// Brief: Master Arm Home Posture
FUNCTION_BLOCK PUBLIC FB_StateCtrlHome EXTENDS FB_MasterArmCtrlBase
VAR_INPUT
END_VAR
VAR_OUTPUT
END_VAR
VAR
	m_homePlanner : FB_TrajMoveJ;
	
	// home motion parameters
	m_homePosture:ARRAY [1..2, 1..7] OF LREAL:=[0.0, -PI/2, 0, -PI, PI, -PI/2, 0,
							 			  			0.0, -PI/2, 0, 0, PI, PI/2, 0];
	m_homeMaxjntVel:Vec7d:=[1.0, 1.0, 1.0, 1.0, 1.0, 1.0, 1.0];
	m_homeMaxjntAcc:Vec7d:=[1.0, 1.0, 1.0, 2.0, 2.0, 2.0, 2.0];
	m_homeMaxjntJerk:Vec7d:=[7(4.0)];
	
	m_endJntPos : Vec7d;
END_VAR

// override this function in each exact controller
METHOD PROTECTED calcCmdJntPos : BOOL
VAR_IN_OUT CONSTANT
	i_slaveIdx :INT;
	i_shoulderPose :ST_Frame;
	i_masterArm :FB_MasterArm;
	i_slaveStatus :ST_SlaveStatus;
END_VAR
VAR 
	i :INT;
	curJntVel :Vec7d;
	curJntPos :Vec7d;
	posErr:Vec7d;
END_VAR
// check if planner is ready
IF m_homePlanner.isGene = FALSE THEN
	calcCmdJntPos:=FALSE;
	RETURN;
END_IF

// traj plan
calcCmdJntPos :=m_homePlanner.evaluate(m_timePeriod, jntPos=> m_cmdJntPos, jntVel=>m_cmdJntVel, jntAcc=> m_cmdJntAcc);

// check if to terminate
curJntVel :=i_masterArm.curJntVel;
curJntPos := i_masterArm.curJntPos;
vecSub(curJntPos,m_endJntPos,posErr);
m_isFinished :=m_timePeriod > m_homePlanner.duration  AND norm(curJntVel)<7*g_jntStaticVelThres AND norm(posErr)<7*g_jntCtrlAngTolLow;
END_METHOD

METHOD PUBLIC init : BOOL
VAR_IN_OUT CONSTANT
	i_masterArm	:FB_MasterArm;
END_VAR
VAR_IN_OUT 
	r_masterArmCtrlCmd :ST_ArmCtrlCmds;
END_VAR

VAR
	i,j :INT;
	startJntPos :Vec7d;
END_VAR
SUPER^.Init(i_masterArm,r_masterArmCtrlCmd);

// traj plan
startJntPos:=i_masterArm.curJntPos;
FOR j:=1 TO 7 DO 
m_endJntPos[j]:=m_homePosture[i_masterArm.armIdx,j];
END_FOR
m_homePlanner.init(startJntPos,m_endJntPos,m_homeMaxjntVel,m_homeMaxjntAcc,m_homeMaxjntJerk);

// update commands to arm
copyCmds(r_masterArmCtrlCmd);
END_METHOD

END_FUNCTION_BLOCK

(* stored: Version 1.1.0.1, ProductVersion 3.1.4024.11
   POU FB_StateCtrlHome: Id {ff8ccb3f-4929-4315-b540-e9546f2dbd07}, SpecialFunc None
   Method calcCmdJntPos: Id {ffa3dbdd-63a1-4101-8d26-d1f3e6e5e2be}
   Method init: Id {c6523e12-84cb-49f8-843e-9a168bb4ce28} *)
